	        20:  // Set Positioning activ?
	            IF "gtyp_HBW".x_Start_Park_Position AND NOT "gtyp_HBW".x_Park_Position_Reached THEN
	                "gtyp_HBW".Horizontal_Axis.x_Start_Positioning := FALSE;
	                "gtyp_HBW".Vertical_Axis.x_Start_Positioning := FALSE;
	                "gtyp_HBW".Horizontal_Axis.x_Reference := FALSE;
	                "gtyp_HBW".Vertical_Axis.x_Reference := FALSE;
	                "QX_HBW_M4_CantileverBackward_Q8" := FALSE;
	                "QX_HBW_M4_CantileverForward_Q7" := FALSE;
	                #li_StepCase := 30;
	            END_IF;

	        30: // homing vertical axis
	            "gtyp_HBW".Vertical_Axis.x_Reference := TRUE;

	            IF NOT "gtyp_HBW".Vertical_Axis.x_Referenced THEN
	                #li_StepCase := 40;
	            END_IF;

	        40: // homed vertical axis
	            IF "gtyp_HBW".Vertical_Axis.x_Referenced THEN
	                "gtyp_HBW".Vertical_Axis.x_Reference := FALSE;
	                #li_StepCase := 50;
	            END_IF;

	        50: // homing horizontal axis
	            "gtyp_HBW".Horizontal_Axis.x_Reference := TRUE;

	            IF NOT "gtyp_HBW".Horizontal_Axis.x_Referenced THEN
	                #li_StepCase := 60;
	            END_IF;

	        60: // homed horizontal axis
	            IF "gtyp_HBW".Horizontal_Axis.x_Referenced THEN
	                "gtyp_HBW".Horizontal_Axis.x_Reference := FALSE;
	                #li_StepCase := 70;
	            END_IF;

	        70: // Position horizontal Axis
	            "gtyp_HBW".Horizontal_Axis.di_Target_Position := "gtyp_HBW".di_Pos_Park_Horizontal;
	            "gtyp_HBW".Horizontal_Axis.x_Start_Positioning := TRUE;

	            IF ("gtyp_HBW".Horizontal_Axis.di_Actual_Position <= ("gtyp_HBW".di_Pos_Park_Horizontal + "gtyp_HBW".Horizontal_Axis.Config.di_Pos_Window))
	                AND ("gtyp_HBW".Horizontal_Axis.di_Actual_Position >= ("gtyp_HBW".di_Pos_Park_Horizontal - "gtyp_HBW".Horizontal_Axis.Config.di_Pos_Window))
	                AND "gtyp_HBW".Horizontal_Axis.x_Position_Reached THEN
	                "gtyp_HBW".Horizontal_Axis.x_Start_Positioning := FALSE;
	                #li_StepCase := 80;
	            END_IF;

	        80: // Position vertical Axis
	            "gtyp_HBW".Vertical_Axis.di_Target_Position := "gtyp_HBW".di_Pos_Park_Vertical;
	            "gtyp_HBW".Vertical_Axis.x_Start_Positioning := TRUE;

	            IF ("gtyp_HBW".Vertical_Axis.di_Actual_Position <= ("gtyp_HBW".di_Pos_Park_Vertical + "gtyp_HBW".Vertical_Axis.Config.di_Pos_Window))
	                AND ("gtyp_HBW".Vertical_Axis.di_Actual_Position >= ("gtyp_HBW".di_Pos_Park_Vertical - "gtyp_HBW".Vertical_Axis.Config.di_Pos_Window))
	                AND "gtyp_HBW".Vertical_Axis.x_Position_Reached THEN
	                "gtyp_HBW".Vertical_Axis.x_Start_Positioning := FALSE;
	                #li_StepCase := 90;
	            END_IF;

	        90: // Deciding which doing
	            "gtyp_HBW".x_Park_Position_Reached := TRUE;


	            // Statement section ELSE
	        ELSE
	            ;
	    END_CASE;

	ELSE
	    #lx_Init := TRUE;
	END_IF;
END_FUNCTION_BLOCK

FUNCTION_BLOCK "PRG_HBW_Axis_Vertical"
TITLE = Program Axis vertical HBW
{ S7_Optimized_Access := 'TRUE' }
AUTHOR : 'A.Schaefer'
VERSION : 0.0
   VAR
      lx_Init { ExternalAccessible := 'False'; ExternalVisible := 'False'; ExternalWritable := 'False'} : Bool;
      lfb_Vertical_Axis { ExternalAccessible := 'False'; ExternalVisible := 'False'; ExternalWritable := 'False'; S7_SetPoint := 'False'} : "FB_Axis";
   END_VAR


BEGIN
	IF #lx_Init THEN

	    // FB Axis vertical
	    #lfb_Vertical_Axis(ini_Axis := 7,
	                       indi_Increment := "gtyp_HBW".Vertical_Axis.di_Increment,
	                       inx_Ref_Switch := "IX_HBW_RefSwitchVerticalAxis_I4",
	                       inx_Referencing := "gtyp_HBW".Vertical_Axis.x_Reference,
	                       inx_Start_Positioning := "gtyp_HBW".Vertical_Axis.x_Start_Positioning,
	                       indi_Target_Position := "gtyp_HBW".Vertical_Axis.di_Target_Position,
	                       ini_PWM := "gtyp_HBW".Vertical_Axis.i_PWM,
	                       inouttyp_Config := "gtyp_HBW".Vertical_Axis.Config,
	                       inouttyp_Setup := "gtyp_SetupAxis");

	    "QX_HBW_M3_VerticalAxisDownward_Q5" := #lfb_Vertical_Axis.outx_Motor_Pos;
	    "QX_HBW_M3_VerticalAxisUpward_Q6" := #lfb_Vertical_Axis.outx_Motor_Neg;
	    "QW_HBW_PWM_VerticalAxis_M3" := #lfb_Vertical_Axis.outi_Motor_PWM;
	    "gtyp_HBW".Vertical_Axis.di_Actual_Position := #lfb_Vertical_Axis.outdi_Actual_Position;
	    "gtyp_HBW".Vertical_Axis.x_Referenced := #lfb_Vertical_Axis.outx_Referenced;
	    "gtyp_HBW".Vertical_Axis.x_Position_Reached := #lfb_Vertical_Axis.outx_Position_Reached;
	ELSE
	    #lx_Init := TRUE;
	END_IF;
END_FUNCTION_BLOCK

FUNCTION_BLOCK "PRG_SLD_Set_Counter_Values"
TITLE = Program Set counter Values SLD
{ S7_Optimized_Access := 'TRUE' }
AUTHOR : 'A.Schaefer'
VERSION : 0.0
   VAR
      lx_Init { ExternalAccessible := 'False'; ExternalVisible := 'False'; ExternalWritable := 'False'} : Bool;
      lfb_R_Trig_Calib_activ {InstructionName := 'R_TRIG'; LibVersion := '1.0'; ExternalAccessible := 'False'; ExternalVisible := 'False'; ExternalWritable := 'False'; S7_SetPoint := 'False'} : R_TRIG;
   END_VAR


BEGIN
	IF #lx_Init THEN

	    // Reload act. Counter Values
	    IF NOT "gtyp_Setup".x_Counter_Value_Calibration THEN
	        "gtyp_Setup".i_Calib_CounterValue_Blue := "gtyp_SLD".i_CounterValue_Blue;
	        "gtyp_Setup".i_Calib_CounterValue_Red := "gtyp_SLD".i_CounterValue_Red;
	        "gtyp_Setup".i_Calib_CounterValue_White := "gtyp_SLD".i_CounterValue_White;
	    END_IF;

	    // Set Counter Values
	    IF "gtyp_Setup".x_Set_CounterValues AND "gtyp_Setup".x_Counter_Value_Calibration THEN
	        "gtyp_SLD".i_CounterValue_Blue := "gtyp_Setup".i_Calib_CounterValue_Blue;
	        "gtyp_SLD".i_CounterValue_Red := "gtyp_Setup".i_Calib_CounterValue_Red;
	        "gtyp_SLD".i_CounterValue_White := "gtyp_Setup".i_Calib_CounterValue_White;
	        "gtyp_Setup".x_Set_CounterValues := FALSE;
	    END_IF;

	ELSE
	    #lx_Init := TRUE;
	END_IF;
END_FUNCTION_BLOCK

FUNCTION_BLOCK "PRG_SLD_Ablauf"
TITLE = Program Ablauf SLD
{ S7_Optimized_Access := 'TRUE' }
AUTHOR : 'A.Schaefer'
VERSION : 0.0
   VAR
      lx_Init { ExternalAccessible := 'False'; ExternalVisible := 'False'; ExternalWritable := 'False'} : Bool;
      lx_Start_TON_Wait { ExternalAccessible := 'False'; ExternalVisible := 'False'; ExternalWritable := 'False'} : Bool;
      lx_Time_Error { ExternalAccessible := 'False'; ExternalVisible := 'False'; ExternalWritable := 'False'} : Bool;
      lt_TON_Wait { ExternalAccessible := 'False'; ExternalVisible := 'False'; ExternalWritable := 'False'} : Time;
      lx_Start_TON_State { ExternalAccessible := 'False'; ExternalVisible := 'False'; ExternalWritable := 'False'} : Bool;
      ldt_MQTT { ExternalAccessible := 'False'; ExternalVisible := 'False'; ExternalWritable := 'False'} : Date_And_Time;
      li_Return_LDT { ExternalAccessible := 'False'; ExternalVisible := 'False'; ExternalWritable := 'False'} : Int;
      li_Lights { ExternalAccessible := 'False'; ExternalVisible := 'False'; ExternalWritable := 'False'} : Int;
      li_Lights_old { ExternalAccessible := 'False'; ExternalVisible := 'False'; ExternalWritable := 'False'} : Int;
      lw_ColorValueMin { ExternalAccessible := 'False'; ExternalVisible := 'False'; ExternalWritable := 'False'} : Word;
      li_CounterActual { ExternalAccessible := 'False'; ExternalVisible := 'False'; ExternalWritable := 'False'} : Int;
      lx_White { ExternalAccessible := 'False'; ExternalVisible := 'False'; ExternalWritable := 'False'} : Bool;
      lx_Blue { ExternalAccessible := 'False'; ExternalVisible := 'False'; ExternalWritable := 'False'} : Bool;
      lx_Red { ExternalAccessible := 'False'; ExternalVisible := 'False'; ExternalWritable := 'False'} : Bool;
      li_StepCase { ExternalAccessible := 'False'; ExternalVisible := 'False'; ExternalWritable := 'False'} : Int;
      ls_Color { ExternalAccessible := 'False'; ExternalVisible := 'False'; ExternalWritable := 'False'} : String;
      lfb_TOF_ConveyerBelt_Out {InstructionName := 'TOF_TIME'; LibVersion := '1.0'; ExternalAccessible := 'False'; ExternalVisible := 'False'; ExternalWritable := 'False'; S7_SetPoint := 'False'} : TOF_TIME;
      lfb_TON_Wait {InstructionName := 'TON_TIME'; LibVersion := '1.0'; ExternalAccessible := 'False'; ExternalVisible := 'False'; ExternalWritable := 'False'; S7_SetPoint := 'False'} : TON_TIME;
      lfb_TON_Error {InstructionName := 'TON_TIME'; LibVersion := '1.0'; ExternalAccessible := 'False'; ExternalVisible := 'False'; ExternalWritable := 'False'; S7_SetPoint := 'False'} : TON_TIME;
      lfb_TON_State {InstructionName := 'TON_TIME'; LibVersion := '1.0'; ExternalAccessible := 'False'; ExternalVisible := 'False'; ExternalWritable := 'False'; S7_SetPoint := 'False'} : TON_TIME;
      lfb_F_Trig_Counter {InstructionName := 'F_TRIG'; LibVersion := '1.0'; ExternalAccessible := 'False'; ExternalVisible := 'False'; ExternalWritable := 'False'; S7_SetPoint := 'False'} : F_TRIG;
      lfb_R_Trig_Counter {InstructionName := 'R_TRIG'; LibVersion := '1.0'; ExternalAccessible := 'False'; ExternalVisible := 'False'; ExternalWritable := 'False'; S7_SetPoint := 'False'} : R_TRIG;
   END_VAR


BEGIN
	IF #lx_Init THEN

	    // Restart after set Positioning
	    IF "gtyp_Setup".x_Color_Sensor_Calibration THEN
	        #li_StepCase := 0;
	    END_IF;

	    // wait time state
	    #lfb_TON_State(IN := NOT #lx_Start_TON_State,
	                   PT := T#2s);

	    // state of the SLD cyclically transmitted to the cloud
	    IF (#lfb_TON_State.Q OR (#li_Lights <> #li_Lights_old)) AND NOT #lx_Start_TON_State THEN
	        #li_Lights_old := #li_Lights;
	        #lx_Start_TON_State := TRUE;
	        #li_Return_LDT := RD_SYS_T(#ldt_MQTT);
	        "gtyp_Interface_Dashboard".Subscribe.State_SLD.ldt_ts := DT_TO_LDT(#ldt_MQTT);
	        "gtyp_Interface_Dashboard".Subscribe.State_SLD.i_code := #li_Lights;
	        "gtyp_Interface_Dashboard".Subscribe.State_SLD.s_description := '';
	        "gtyp_Interface_Dashboard".Subscribe.State_SLD.s_station := 'sld';
	        "gtyp_Interface_Dashboard".Subscribe.State_SLD.s_target := '';
	    END_IF;

	    // restart wait time state
	    IF NOT #lfb_TON_State.Q AND #lx_Start_TON_State THEN
	        #lx_Start_TON_State := FALSE;
	    END_IF;

	    // FB TON Wait
	    #lfb_TON_Wait(IN := #lx_Start_TON_Wait,
	                  PT := #lt_TON_Wait);

	    // runtime monitoring error
	    #lfb_TON_Error(IN := #lx_Time_Error,
	                   PT := T#30s);

	    // rising edge pulse counter
	    #lfb_R_Trig_Counter(CLK := "IX_SLD_PulseCounter_I1");

	    // falling edge pulse counter
	    #lfb_F_Trig_Counter(CLK := "IX_SLD_PulseCounter_I1");

	    // step chain SLD
	    CASE #li_StepCase OF

	        0:  // Init
	            #lx_Start_TON_Wait := FALSE;
	            #lx_Time_Error := FALSE;
	            #li_Lights := 1;

	            IF NOT "gtyp_SLD".x_Error AND NOT "gtyp_Setup".x_Color_Sensor_Calibration THEN
	                #li_StepCase := 10;
	            END_IF;

	        10: // turn-on Compressor and wait sequence
	            #li_Lights := 2;
	            "QX_SLD_Compressor_Q2" := TRUE;

	            #lx_Start_TON_Wait := TRUE;
	            #lt_TON_Wait := T#1000ms;

	            IF #lfb_TON_Wait.Q THEN
	                #lx_Start_TON_Wait := FALSE;
	                #li_StepCase := 20;
	            END_IF;

	        20:  // reset Ejectors
	            "QX_SLD_ValveFirstEjectorWhite_Q3" := FALSE;
	            "QX_SLD_ValveSecondEjectorRed_Q4" := FALSE;
	            "QX_SLD_ValveThirdEjectorBlue_Q5" := FALSE;
	            "QX_SLD_M1_ConveyorBelt_Q1" := FALSE;

	            #lx_Start_TON_Wait := TRUE;
	            #lt_TON_Wait := T#2000ms;

	            IF #lfb_TON_Wait.Q THEN
	                #lx_Start_TON_Wait := FALSE;
	                #li_StepCase := 30;
	            END_IF;

	        30: // turn-off Compressor

	            "QX_SLD_Compressor_Q2" := FALSE;

	            #li_StepCase := 40;

	        40: // start belt if Light barrier I2 active

	            #li_Lights := 1;
	            IF NOT "IX_SLD_LightBarrierInlet_I2" THEN
	                "gtyp_Interface_Dashboard".Subscribe.State_SLD.x_active := TRUE;
	                #li_Lights := 2;
	                "QX_SLD_Compressor_Q2" := TRUE;
	                "QX_SLD_M1_ConveyorBelt_Q1" := TRUE;
	                #lw_ColorValueMin := 40000;
	                #li_CounterActual := 0;
	                #lx_Blue := FALSE;
	                #lx_Red := FALSE;
	                #lx_White := FALSE;
	                #li_StepCase := 50;
	            END_IF;

	        50: // take the min Value of the Color sensor
	            IF #lw_ColorValueMin > "IW_SLD_ColorSensor_A4" THEN
	                #lw_ColorValueMin := "IW_SLD_ColorSensor_A4";
	            END_IF;

	            #lx_Time_Error := TRUE;

	            // Stop when light barrier I3 on
	            IF NOT "IX_SLD_LightBarrierBehindColorSensor_I3" THEN
	                #lx_Time_Error := FALSE;
	                #li_StepCase := 60;
	            END_IF;

	            // runtime error
	            IF #lfb_TON_Error.Q THEN
	                #li_Lights := 4;
	                #lx_Time_Error := FALSE;
	                "QX_SLD_Compressor_Q2" := FALSE;
	                "QX_SLD_M1_ConveyorBelt_Q1" := FALSE;
	                "gtyp_Interface_Dashboard".Subscribe.State_SLD.x_active := FALSE;
	                "gtyp_SLD".x_Error := TRUE;
	                #li_StepCase := 0;
	            END_IF;

	        60: // analyze color

	            IF #lw_ColorValueMin >= "gtyp_SLD".w_Threshold_Red_Blue THEN
	                #lx_Blue := TRUE;
	            ELSIF #lw_ColorValueMin <= "gtyp_SLD".w_Threshold_White_Red THEN
	                #lx_White := TRUE;
	            ELSIF #lw_ColorValueMin > "gtyp_SLD".w_Threshold_White_Red AND #lw_ColorValueMin < "gtyp_SLD".w_Threshold_Red_Blue THEN
	                #lx_Red := TRUE;
	            END_IF;

	            // actual counter
	            IF #lfb_R_Trig_Counter.Q OR #lfb_F_Trig_Counter.Q THEN
	                #li_CounterActual := #li_CounterActual + 1;
	            END_IF;

	            // Reached counter value and color set Ejector
	            IF (#li_CounterActual = "gtyp_SLD".i_CounterValue_Blue) AND #lx_Blue THEN
	                "QX_SLD_ValveThirdEjectorBlue_Q5" := TRUE;
	                #li_Return_LDT := RD_SYS_T(#ldt_MQTT);
	                "gtyp_SLD".Workpiece.s_state := 'PROCESSED';
	                "gtyp_SLD".History[7].i_code := 700;
	                "gtyp_SLD".History[7].ldt_ts := DT_TO_LDT(#ldt_MQTT);
	                #li_StepCase := 70;
	            ELSIF (#li_CounterActual = "gtyp_SLD".i_CounterValue_White) AND #lx_White THEN
	                "QX_SLD_ValveFirstEjectorWhite_Q3" := TRUE;
	                #li_Return_LDT := RD_SYS_T(#ldt_MQTT);
	                "gtyp_SLD".Workpiece.s_state := 'PROCESSED';
	                "gtyp_SLD".History[7].i_code := 700;
	                "gtyp_SLD".History[7].ldt_ts := DT_TO_LDT(#ldt_MQTT);
	                #li_StepCase := 70;
	            ELSIF (#li_CounterActual = "gtyp_SLD".i_CounterValue_Red) AND #lx_Red THEN
	                "QX_SLD_ValveSecondEjectorRed_Q4" := TRUE;
	                #li_Return_LDT := RD_SYS_T(#ldt_MQTT);
	                "gtyp_SLD".Workpiece.s_state := 'PROCESSED';
	                "gtyp_SLD".History[7].i_code := 700;
	                "gtyp_SLD".History[7].ldt_ts := DT_TO_LDT(#ldt_MQTT);
	                #li_StepCase := 70;
	            ELSIF (#li_CounterActual = 80) THEN
	                #li_Lights := 4;
	                "gtyp_SLD".x_Error := TRUE;
	                #li_StepCase := 70;
	            END_IF;

	        70: // wait sequence
	            #lx_Start_TON_Wait := TRUE;
	            #lt_TON_Wait := T#500ms;

	            IF #lfb_TON_Wait.Q THEN
	                "QX_SLD_ValveThirdEjectorBlue_Q5" := FALSE;
	                "QX_SLD_ValveFirstEjectorWhite_Q3" := FALSE;
	                "QX_SLD_ValveSecondEjectorRed_Q4" := FALSE;
	                #lx_Start_TON_Wait := FALSE;
	                #li_StepCase := 80;
	            END_IF;

	        80: // wait sequence

	            #lx_Start_TON_Wait := TRUE;
	            #lt_TON_Wait := T#2000ms;

	            IF #lfb_TON_Wait.Q THEN
	                "QX_SLD_Compressor_Q2" := FALSE;
	                #lx_Start_TON_Wait := FALSE;
	                #li_StepCase := 90;
	            END_IF;

	        90: // Stop belt
	            "QX_SLD_M1_ConveyorBelt_Q1" := FALSE;
	            #li_StepCase := 40;
	            // Statement section ELSE
	        ELSE
	            ;
	    END_CASE;

	ELSE
	    "gtyp_SLD".x_Error := FALSE;
	    #li_Lights := 1;
	    #lx_Init := TRUE;
	END_IF;
END_FUNCTION_BLOCK

FUNCTION_BLOCK "PRG_HBW_Axis_Horizontal"
TITLE = Program Axis horizontal HBW
{ S7_Optimized_Access := 'TRUE' }
AUTHOR : 'A.Schaefer'
VERSION : 0.0
   VAR
      lx_Init { ExternalAccessible := 'False'; ExternalVisible := 'False'; ExternalWritable := 'False'} : Bool;
      lfb_Horizontal_Axis { ExternalAccessible := 'False'; ExternalVisible := 'False'; ExternalWritable := 'False'; S7_SetPoint := 'False'} : "FB_Axis";
   END_VAR


BEGIN
	IF #lx_Init THEN

	    // FB Axis horizontal
	    #lfb_Horizontal_Axis(ini_Axis := 6,
	                         indi_Increment := "gtyp_HBW".Horizontal_Axis.di_Increment,
	                         inx_Ref_Switch := "IX_HBW_RefSwitchHorizontalAxis_I1",
	                         inx_Referencing := "gtyp_HBW".Horizontal_Axis.x_Reference,
	                         inx_Start_Positioning := "gtyp_HBW".Horizontal_Axis.x_Start_Positioning,
	                         indi_Target_Position := "gtyp_HBW".Horizontal_Axis.di_Target_Position,
	                         ini_PWM := "gtyp_HBW".Horizontal_Axis.i_PWM,
	                         inouttyp_Config := "gtyp_HBW".Horizontal_Axis.Config,
	                         inouttyp_Setup := "gtyp_SetupAxis");

	    "QX_HBW_M2_HorizontalTowardsRack_Q3" := #lfb_Horizontal_Axis.outx_Motor_Pos;
	    "QX_HBW_M2_HorizontalTowardsConveyorBelt_Q4" := #lfb_Horizontal_Axis.outx_Motor_Neg;
	    "QW_HBW_PWM_HorizontalAxis_M2" := #lfb_Horizontal_Axis.outi_Motor_PWM;
	    "gtyp_HBW".Horizontal_Axis.di_Actual_Position := #lfb_Horizontal_Axis.outdi_Actual_Position;
	    "gtyp_HBW".Horizontal_Axis.x_Referenced := #lfb_Horizontal_Axis.outx_Referenced;
	    "gtyp_HBW".Horizontal_Axis.x_Position_Reached := #lfb_Horizontal_Axis.outx_Position_Reached;
	ELSE
	    #lx_Init := TRUE;
	END_IF;
END_FUNCTION_BLOCK

FUNCTION_BLOCK "PRG_SLD_Calibration_Color"
TITLE = Program Calibration Color Sensor SLD
{ S7_Optimized_Access := 'TRUE' }
AUTHOR : 'A.Schaefer'
VERSION : 0.0
   VAR
      lx_Init { ExternalAccessible := 'False'; ExternalVisible := 'False'; ExternalWritable := 'False'} : Bool;
      lx_Start_TON_Wait { ExternalAccessible := 'False'; ExternalVisible := 'False'; ExternalWritable := 'False'} : Bool;
      lx_Start_Positioning_m { ExternalAccessible := 'False'; ExternalVisible := 'False'; ExternalWritable := 'False'} : Bool;
      lt_TON_Wait { ExternalAccessible := 'False'; ExternalVisible := 'False'; ExternalWritable := 'False'} : Time;
      li_StepCase { ExternalAccessible := 'False'; ExternalVisible := 'False'; ExternalWritable := 'False'} : Int;
      lw_ColorValueMin { ExternalAccessible := 'False'; ExternalVisible := 'False'; ExternalWritable := 'False'} : Word;
      ldi_Pos_Horizontal { ExternalAccessible := 'False'; ExternalVisible := 'False'; ExternalWritable := 'False'} : DInt;
      ldi_Pos_Vertical { ExternalAccessible := 'False'; ExternalVisible := 'False'; ExternalWritable := 'False'} : DInt;
      lfb_R_Trig_Deaktivate {InstructionName := 'R_TRIG'; LibVersion := '1.0'; ExternalAccessible := 'False'; ExternalVisible := 'False'; ExternalWritable := 'False'; S7_SetPoint := 'False'} : R_TRIG;
      lfb_TON_Wait {InstructionName := 'TON_TIME'; LibVersion := '1.0'; ExternalAccessible := 'False'; ExternalVisible := 'False'; ExternalWritable := 'False'; S7_SetPoint := 'False'} : TON_TIME;
   END_VAR


BEGIN
	IF #lx_Init THEN

	    // FB TON Wait
	    #lfb_TON_Wait(IN := #lx_Start_TON_Wait,
	                  PT := #lt_TON_Wait);

	    #lfb_R_Trig_Deaktivate(CLK := NOT "gtyp_Setup".x_Color_Sensor_Calibration
	                           OR NOT ("gtyp_Setup".i_Color_Sensor_Selection = 2));
	    // Deaktivate step 0
	    IF #lfb_R_Trig_Deaktivate.Q THEN
	        "gtyp_Setup".x_Calculate_Value_Color := FALSE;
	        "gtyp_Setup".x_Set_Calib_Value_Color_Blue := FALSE;
	        "gtyp_Setup".x_Set_Calib_Value_Color_Red := FALSE;
	        "gtyp_Setup".x_Set_Calib_Value_Color_White := FALSE;
	        "gtyp_Setup".w_Calib_ColorValue_Blue := 0;
	        "gtyp_Setup".w_Calib_ColorValue_Red := 0;
	        "gtyp_Setup".w_Calib_ColorValue_White := 0;
	        "gtyp_Setup".w_Threshold_Red_Blue := 0;
	        "gtyp_Setup".w_Threshold_White_Red := 0;
	        "QX_SLD_M1_ConveyorBelt_Q1" := FALSE;
	        #lw_ColorValueMin := 16#FF;
	        #li_StepCase := 0;
	    END_IF;

	    // step chain HBW
	    CASE #li_StepCase OF

	        0:  // init
	            #lx_Start_TON_Wait := FALSE;
	            #li_StepCase := 10;

	        10:  // Set Calibration activ?
	            IF "gtyp_Setup".x_Color_Sensor_Calibration
	                AND ("gtyp_Setup".i_Color_Sensor_Selection = 2) THEN
	                "gtyp_Setup".x_Calculate_Value_Color := FALSE;
	                "gtyp_Setup".x_Set_Calib_Value_Color_Blue := FALSE;
	                "gtyp_Setup".x_Set_Calib_Value_Color_Red := FALSE;
	                "gtyp_Setup".x_Set_Calib_Value_Color_White := FALSE;
	                "gtyp_Setup".w_Calib_ColorValue_Blue := 0;
	                "gtyp_Setup".w_Calib_ColorValue_Red := 0;
	                "gtyp_Setup".w_Calib_ColorValue_White := 0;
	                "gtyp_Setup".w_Threshold_Red_Blue := 0;
	                "gtyp_Setup".w_Threshold_White_Red := 0;
	                "QX_SLD_M1_ConveyorBelt_Q1" := FALSE;
	                #lw_ColorValueMin := 16#FFFF;
	                #li_StepCase := 20;
	            END_IF;

	        20: // wait for set Values or Calculate

	            IF NOT "IX_SLD_LightBarrierInlet_I2" THEN
	                "QX_SLD_M1_ConveyorBelt_Q1" := TRUE;
	                #lw_ColorValueMin := 16#FFFF;
	            END_IF;

	            IF #lw_ColorValueMin > "IW_SLD_ColorSensor_A4" THEN
	                #lw_ColorValueMin := "IW_SLD_ColorSensor_A4";
	            END_IF;

	            IF NOT "IX_SLD_LightBarrierBehindColorSensor_I3" THEN
	                "QX_SLD_M1_ConveyorBelt_Q1" := FALSE;
	            END_IF;

	            // Start new Positioning
	            IF "gtyp_Setup".x_Set_Calib_Value_Color_Blue THEN
	                "gtyp_Setup".w_Calib_ColorValue_Blue := #lw_ColorValueMin;
	                "gtyp_Setup".x_Set_Calib_Value_Color_Blue := FALSE;
	            ELSIF "gtyp_Setup".x_Set_Calib_Value_Color_Red THEN
	                "gtyp_Setup".w_Calib_ColorValue_Red := #lw_ColorValueMin;
	                "gtyp_Setup".x_Set_Calib_Value_Color_Red := FALSE;
	            ELSIF "gtyp_Setup".x_Set_Calib_Value_Color_White THEN
	                "gtyp_Setup".w_Calib_ColorValue_White := #lw_ColorValueMin;
	                "gtyp_Setup".x_Set_Calib_Value_Color_White := FALSE;
	            END_IF;

	            "gtyp_Setup".w_Threshold_White_Red := "gtyp_Setup".w_Calib_ColorValue_White + (("gtyp_Setup".w_Calib_ColorValue_Red - "gtyp_Setup".w_Calib_ColorValue_White) / 2);
	            "gtyp_Setup".w_Threshold_Red_Blue := "gtyp_Setup".w_Calib_ColorValue_Red + (("gtyp_Setup".w_Calib_ColorValue_Blue - "gtyp_Setup".w_Calib_ColorValue_Red) / 2);

	            IF "gtyp_Setup".x_Calculate_Value_Color THEN
	                "gtyp_SLD".w_Threshold_White_Red := "gtyp_Setup".w_Threshold_White_Red;
	                "gtyp_SLD".w_Threshold_Red_Blue := "gtyp_Setup".w_Threshold_Red_Blue;
	                "gtyp_Setup".x_Calculate_Value_Color := FALSE;
	            END_IF;

	            // Statement section ELSE
	        ELSE
	            ;
	    END_CASE;

	    IF ("gtyp_Setup".i_Color_Sensor_Selection = 2) THEN
	        // Reload Pos Value
	        "gtyp_Setup".w_Actual_ColorValue := "IW_SLD_ColorSensor_A4";
	    END_IF;
	ELSE
	    #lx_Init := TRUE;
	END_IF;
END_FUNCTION_BLOCK

FUNCTION_BLOCK "PRG_DSO_Status"
TITLE = Program Status DSO
{ S7_Optimized_Access := 'TRUE' }
AUTHOR : 'A.Schaefer'
VERSION : 0.0
   VAR
      lx_Init { ExternalAccessible := 'False'; ExternalVisible := 'False'; ExternalWritable := 'False'} : Bool;
      lx_Start { ExternalAccessible := 'False'; ExternalVisible := 'False'; ExternalWritable := 'False'} : Bool;
      li_StepCase { ExternalAccessible := 'False'; ExternalVisible := 'False'; ExternalWritable := 'False'} : Int;
      ldt_MQTT { ExternalAccessible := 'False'; ExternalVisible := 'False'; ExternalWritable := 'False'} : Date_And_Time;
      li_Return_LDT { ExternalAccessible := 'False'; ExternalVisible := 'False'; ExternalWritable := 'False'} : Int;
      li_code_old { ExternalAccessible := 'False'; ExternalVisible := 'False'; ExternalWritable := 'False'} : Int;
      lfb_R_Trig_Outsourcing {InstructionName := 'R_TRIG'; LibVersion := '1.0'; ExternalAccessible := 'False'; ExternalVisible := 'False'; ExternalWritable := 'False'; S7_SetPoint := 'False'} : R_TRIG;
      lfb_R_Trig_Take_Workpiece {InstructionName := 'R_TRIG'; LibVersion := '1.0'; ExternalAccessible := 'False'; ExternalVisible := 'False'; ExternalWritable := 'False'; S7_SetPoint := 'False'} : R_TRIG;
      lfb_TON_Status {InstructionName := 'TON_TIME'; LibVersion := '1.0'; ExternalAccessible := 'False'; ExternalVisible := 'False'; ExternalWritable := 'False'; S7_SetPoint := 'False'} : TON_TIME;
      lfb_TON_End_Order {InstructionName := 'TON_TIME'; LibVersion := '1.0'; ExternalAccessible := 'False'; ExternalVisible := 'False'; ExternalWritable := 'False'; S7_SetPoint := 'False'} : TON_TIME;
      lx_StartStatus { ExternalAccessible := 'False'; ExternalVisible := 'False'; ExternalWritable := 'False'} : Bool;
      lx_StartEndOrder { ExternalAccessible := 'False'; ExternalVisible := 'False'; ExternalWritable := 'False'} : Bool;
      lx_StartTimer { ExternalAccessible := 'False'; ExternalVisible := 'False'; ExternalWritable := 'False'} : Bool;
   END_VAR


BEGIN
	IF #lx_Init THEN

	    // wait time state
	    #lfb_TON_Status(IN := NOT #lx_StartStatus,
	                    PT := T#2s);

	    // rising/falling edge light barrier DSI
	    #lfb_R_Trig_Outsourcing(CLK := NOT "IX_SSC_LightBarrierOutsourcing_I4");
	    #lfb_R_Trig_Take_Workpiece(CLK := "IX_SSC_LightBarrierOutsourcing_I4");

	    // start wait time end order
	    IF NOT "IX_SSC_LightBarrierOutsourcing_I4" AND ("gtyp_Interface_Dashboard".Subscribe.State_Order.s_state = 'SHIPPED') THEN
	        #lx_StartEndOrder := TRUE;
	    END_IF;

	    // wait time end order
	    #lfb_TON_End_Order(IN := #lx_StartEndOrder,
	                       PT := T#5s);

	    IF #lfb_R_Trig_Take_Workpiece.Q OR #lfb_TON_End_Order.Q THEN
	        #lx_StartEndOrder := FALSE;
	        "gtyp_Interface_Dashboard".Subscribe.State_Order.ldt_ts := DT_TO_LDT(#ldt_MQTT);
	        "gtyp_Interface_Dashboard".Subscribe.State_Order.s_state := 'WAITING_FOR_ORDER';
	        "gtyp_Interface_Dashboard".Subscribe.State_Order.s_type := '';
	        "gtyp_Interface_Dashboard".Subscribe.State_DSO.x_active := FALSE;
	    END_IF;

	    // state of the DSO transmitted to the cloud
	    IF (#lfb_TON_Status.Q OR #lfb_R_Trig_Outsourcing.Q OR #lfb_R_Trig_Take_Workpiece.Q) AND NOT #lx_StartStatus THEN
	        #lx_StartStatus := TRUE;
	        #li_Return_LDT := RD_SYS_T(#ldt_MQTT);
	        IF NOT "IX_SSC_LightBarrierOutsourcing_I4" THEN
	            "gtyp_Interface_Dashboard".Subscribe.State_DSO.i_code := 0;
	        ELSE
	            "gtyp_Interface_Dashboard".Subscribe.State_DSO.i_code := 1;
	        END_IF;
	        "gtyp_Interface_Dashboard".Subscribe.State_DSO.ldt_ts := DT_TO_LDT(#ldt_MQTT);
	        "gtyp_Interface_Dashboard".Subscribe.State_DSO.s_station := 'dso';
	        "gtyp_Interface_Dashboard".Subscribe.State_DSO.s_target := '';
	        "gtyp_Interface_Dashboard".Subscribe.State_DSO.s_description := '';
	    END_IF;

	    IF NOT #lfb_TON_Status.Q AND #lx_StartStatus THEN
	        #lx_StartStatus := FALSE;
	    END_IF;
	ELSE
	    #lx_Init := TRUE;
	    #lx_StartEndOrder := FALSE;
	END_IF;
END_FUNCTION_BLOCK

DATA_BLOCK "PRG_SLD_Ablauf_DB"
{ S7_Optimized_Access := 'TRUE' }
AUTHOR : 'A.Schaefer'
VERSION : 0.1
NON_RETAIN
"PRG_SLD_Ablauf"

BEGIN

END_DATA_BLOCK

DATA_BLOCK "PRG_SSC_Axis_Horizontal_DB"
{ S7_Optimized_Access := 'TRUE' }
AUTHOR : 'A.Schaefer'
VERSION : 0.1
NON_RETAIN
"PRG_SSC_Axis_Horizontal"

BEGIN

END_DATA_BLOCK

DATA_BLOCK "PRG_SSC_Axis_Vertical_DB"
{ S7_Optimized_Access := 'TRUE' }
AUTHOR : 'A.Schaefer'
VERSION : 0.1
NON_RETAIN
"PRG_SSC_Axis_Vertical"

BEGIN

END_DATA_BLOCK

DATA_BLOCK "PRG_SLD_Calibration_Color_DB"
{ S7_Optimized_Access := 'TRUE' }
AUTHOR : 'A.Schaefer'
VERSION : 0.1
NON_RETAIN
"PRG_SLD_Calibration_Color"

BEGIN

END_DATA_BLOCK

DATA_BLOCK "PRG_SSC_Set_Park_Position_DB"
{ S7_Optimized_Access := 'TRUE' }
AUTHOR : 'A.Schaefer'
VERSION : 0.0
NON_RETAIN
"PRG_SSC_Set_Park_Position"

BEGIN

END_DATA_BLOCK

DATA_BLOCK "PRG_SSC_Light_DB"
{ S7_Optimized_Access := 'TRUE' }
AUTHOR : 'A.Schaefer'
VERSION : 0.1
NON_RETAIN
"PRG_SSC_Light"

BEGIN

END_DATA_BLOCK

DATA_BLOCK "PRG_SLD_Set_Counter_Values_DB"
{ S7_Optimized_Access := 'TRUE' }
AUTHOR : 'A.Schaefer'
VERSION : 0.1
NON_RETAIN
"PRG_SLD_Set_Counter_Values"

BEGIN

END_DATA_BLOCK

DATA_BLOCK "PRG_SSC_Set_Positioning_DB"
{ S7_Optimized_Access := 'TRUE' }
AUTHOR : 'A.Schaefer'
VERSION : 0.1
NON_RETAIN
"PRG_SSC_Set_Positioning"

BEGIN

END_DATA_BLOCK

DATA_BLOCK "PRG_DSI_Status_DB"
{ S7_Optimized_Access := 'TRUE' }
AUTHOR : 'A.Schaefer'
VERSION : 0.1
NON_RETAIN
"PRG_DSI_Status"

BEGIN

END_DATA_BLOCK

DATA_BLOCK "PRG_SSC_Ablauf_DB"
{ S7_Optimized_Access := 'TRUE' }
AUTHOR : 'A.Schaefer'
VERSION : 0.1
NON_RETAIN
"PRG_SSC_Ablauf"

BEGIN

END_DATA_BLOCK

DATA_BLOCK "RT_INFO_scl_OB30"
{ S7_Optimized_Access := 'TRUE' }
VERSION : 0.1
NON_RETAIN
   VAR
      mode { ExternalAccessible := 'False'; ExternalVisible := 'False'; ExternalWritable := 'False'} : UInt;   // Mode 1 = Runtime of a specific OB; 2 = Maximum runtime of a specific OB; 3 = Minimum runtime of a specific OB; 10 = Mean value of the percentage of total runtime used by higher-priority OBs; ...
      obNbr { ExternalAccessible := 'False'; ExternalVisible := 'False'; ExternalWritable := 'False'} : OB_ANY;   // OB to read
      infoData { ExternalAccessible := 'False'; ExternalVisible := 'False'; ExternalWritable := 'False'} : LTime;   // mode 1 --> Runtime in LTIME
      returnValue { ExternalAccessible := 'False'; ExternalVisible := 'False'; ExternalWritable := 'False'} : Int;   // Error information of instruction
   END_VAR


BEGIN
   mode := 1;
   obNbr := 1;

END_DATA_BLOCK

DATA_BLOCK "PRG_SSC_Calibration_Color_DB"
{ S7_Optimized_Access := 'TRUE' }
AUTHOR : 'A.Schaefer'
VERSION : 0.1
NON_RETAIN
"PRG_SSC_Calibration_Color"

BEGIN

END_DATA_BLOCK

DATA_BLOCK "PRG_HBW_Ablauf_DB"
{ S7_Optimized_Access := 'TRUE' }
AUTHOR : 'A.Schaefer'
VERSION : 0.1
NON_RETAIN
"PRG_HBW_Ablauf"

BEGIN

END_DATA_BLOCK

DATA_BLOCK "RT_INFO_scl_OB1"
{ S7_Optimized_Access := 'TRUE' }
VERSION : 0.1
NON_RETAIN
   VAR
      mode { ExternalAccessible := 'False'; ExternalVisible := 'False'; ExternalWritable := 'False'} : UInt;   // Mode 1 = Runtime of a specific OB; 2 = Maximum runtime of a specific OB; 3 = Minimum runtime of a specific OB; 10 = Mean value of the percentage of total runtime used by higher-priority OBs; ...
      obNbr { ExternalAccessible := 'False'; ExternalVisible := 'False'; ExternalWritable := 'False'} : OB_ANY;   // OB to read
      infoData { ExternalAccessible := 'False'; ExternalVisible := 'False'; ExternalWritable := 'False'} : LTime;   // mode 1 --> Runtime in LTIME
      returnValue { ExternalAccessible := 'False'; ExternalVisible := 'False'; ExternalWritable := 'False'} : Int;   // Error information of instruction
   END_VAR


BEGIN
   mode := 1;
   obNbr := 1;

END_DATA_BLOCK

DATA_BLOCK "PRG_MPO_Set_Park_Position_DB"
{ S7_Optimized_Access := 'TRUE' }
AUTHOR : 'A.Schaefer'
VERSION : 0.0
NON_RETAIN
"PRG_MPO_Set_Park_Position"

BEGIN

END_DATA_BLOCK

DATA_BLOCK "PRG_HBW_Set_Park_Position_DB"
{ S7_Optimized_Access := 'TRUE' }
AUTHOR : 'A.Schaefer'
VERSION : 0.0
NON_RETAIN
"PRG_HBW_Set_Park_Position"

BEGIN

END_DATA_BLOCK

DATA_BLOCK "PRG_Acknowledge_DB"
{ S7_Optimized_Access := 'TRUE' }
AUTHOR : 'A.Schaefer'
VERSION : 0.1
NON_RETAIN
"PRG_Acknowledge"

BEGIN

END_DATA_BLOCK

DATA_BLOCK "PRG_HBW_Axis_Vertical_DB"
{ S7_Optimized_Access := 'TRUE' }
AUTHOR : 'A.Schaefer'
VERSION : 0.1
NON_RETAIN
"PRG_HBW_Axis_Vertical"

BEGIN

END_DATA_BLOCK

DATA_BLOCK "PRG_HBW_Axis_Horizontal_DB"
{ S7_Optimized_Access := 'TRUE' }
AUTHOR : 'A.Schaefer'
VERSION : 0.1
NON_RETAIN
"PRG_HBW_Axis_Horizontal"

BEGIN

END_DATA_BLOCK

DATA_BLOCK "PRG_NFC_DB"
{ S7_Optimized_Access := 'TRUE' }
AUTHOR : 'A.Schaefer'
VERSION : 0.1
NON_RETAIN
"PRG_NFC"

BEGIN

END_DATA_BLOCK

DATA_BLOCK "PRG_VGR_Axis_rotate_DB"
{ S7_Optimized_Access := 'TRUE' }
AUTHOR : 'A.Schaefer'
VERSION : 0.1
NON_RETAIN
"PRG_VGR_Axis_rotate"

BEGIN

END_DATA_BLOCK

DATA_BLOCK "PRG_VGR_Ablauf_DB"
{ S7_Optimized_Access := 'TRUE' }
AUTHOR : 'A.Schaefer'
VERSION : 0.1
NON_RETAIN
"PRG_VGR_Ablauf"

BEGIN

END_DATA_BLOCK

DATA_BLOCK "PRG_Order_DB"
{ S7_Optimized_Access := 'TRUE' }
AUTHOR : 'A.Schaefer'
VERSION : 0.1
NON_RETAIN
"PRG_Order"

BEGIN

END_DATA_BLOCK

DATA_BLOCK "PRG_VGR_Axis_horizontal_DB"
{ S7_Optimized_Access := 'TRUE' }
AUTHOR : 'A.Schaefer'
VERSION : 0.1
NON_RETAIN
"PRG_VGR_Axis_horizontal"

BEGIN

END_DATA_BLOCK

DATA_BLOCK "PRG_DSO_Status_DB"
{ S7_Optimized_Access := 'TRUE' }
AUTHOR : 'A.Schaefer'
VERSION : 0.1
NON_RETAIN
"PRG_DSO_Status"

BEGIN

END_DATA_BLOCK

DATA_BLOCK "PRG_VGR_Set_Park_Position_DB"
{ S7_Optimized_Access := 'TRUE' }
AUTHOR : 'A.Schaefer'
VERSION : 0.0
NON_RETAIN
"PRG_VGR_Set_Park_Position"

BEGIN

END_DATA_BLOCK

DATA_BLOCK "PRG_MPO_Ablauf_DB"
{ S7_Optimized_Access := 'TRUE' }
AUTHOR : 'A.Schaefer'
VERSION : 0.1
NON_RETAIN
"PRG_MPO_Ablauf"

BEGIN

END_DATA_BLOCK

DATA_BLOCK "PRG_VGR_Set_Positioning_DB"
{ S7_Optimized_Access := 'TRUE' }
AUTHOR : 'A.Schaefer'
VERSION : 0.1
NON_RETAIN
"PRG_VGR_Set_Positioning"

BEGIN

END_DATA_BLOCK

DATA_BLOCK "PRG_HBW_Set_Positioning_DB"
{ S7_Optimized_Access := 'TRUE' }
AUTHOR : 'A.Schaefer'
VERSION : 0.1
NON_RETAIN
"PRG_HBW_Set_Positioning"

BEGIN

END_DATA_BLOCK

DATA_BLOCK "PRG_VGR_Axis_vertical_DB"
{ S7_Optimized_Access := 'TRUE' }
AUTHOR : 'A.Schaefer'
VERSION : 0.1
NON_RETAIN
"PRG_VGR_Axis_vertical"

BEGIN

END_DATA_BLOCK

ORGANIZATION_BLOCK "Main"
TITLE = "Main Program Sweep (Cycle)"
{ S7_Optimized_Access := 'TRUE' }
AUTHOR : 'A.Schaefer'
VERSION : 0.0

BEGIN
	// current cycle Time OB30
	"RT_INFO_scl_OB30".mode := 1;
	"RT_INFO_scl_OB30".obNbr := 30;
	"RT_INFO_scl_OB30".returnValue := RT_INFO(MODE := "RT_INFO_scl_OB30".mode,
	                                          OB := "RT_INFO_scl_OB30".obNbr,
	                                          INFO := "RT_INFO_scl_OB30".infoData);

	// current cycle Time OB1
	"RT_INFO_scl_OB1".mode := 1;
	"RT_INFO_scl_OB1".obNbr := 1;
	"RT_INFO_scl_OB1".returnValue := RT_INFO(MODE := "RT_INFO_scl_OB1".mode,
	                                         OB := "RT_INFO_scl_OB1".obNbr,
	                                         INFO := "RT_INFO_scl_OB1".infoData);

	// sources SSC
	"PRG_SSC_Ablauf_DB"();
	"PRG_SSC_Set_Positioning_DB"();
	"PRG_SSC_Set_Park_Position_DB"();
	"PRG_SSC_Calibration_Color_DB"();
	"PRG_SSC_Axis_Vertical_DB"();
	"PRG_SSC_Axis_Horizontal_DB"();
	"PRG_SSC_Light_DB"();

	// sources VGR
	"PRG_VGR_Ablauf_DB"();
	"PRG_VGR_Set_Positioning_DB"();
	"PRG_VGR_Set_Park_Position_DB"();
	"PRG_VGR_Axis_horizontal_DB"();
	"PRG_VGR_Axis_vertical_DB"();
	"PRG_VGR_Axis_rotate_DB"();
	"PRG_NFC_DB"();

	// sources HBW
	"PRG_HBW_Ablauf_DB"();
	"PRG_HBW_Set_Positioning_DB"();
	"PRG_HBW_Set_Park_Position_DB"();
	"PRG_HBW_Axis_Vertical_DB"();
	"PRG_HBW_Axis_Horizontal_DB"();

	// sources MPO
	"PRG_MPO_Ablauf_DB"();
	"PRG_MPO_Set_Park_Position_DB"();

	// sources SLD
	"PRG_SLD_Ablauf_DB"();
	"PRG_SLD_Calibration_Color_DB"();
	"PRG_SLD_Set_Counter_Values_DB"();

	// sources input/output
	"PRG_DSI_Status_DB"();
	"PRG_DSO_Status_DB"();

	// sources dashboard
	"PRG_Order_DB"();
	"PRG_Acknowledge_DB"();

END_ORGANIZATION_BLOCK

